(* PLC project Unnamed, Unknown Unnamed 1 *)
(* stored: creationDateTime 2024-02-27T18:06:15, modificationDateTime 2024-02-27T18:24:05 *)

PROGRAM Example

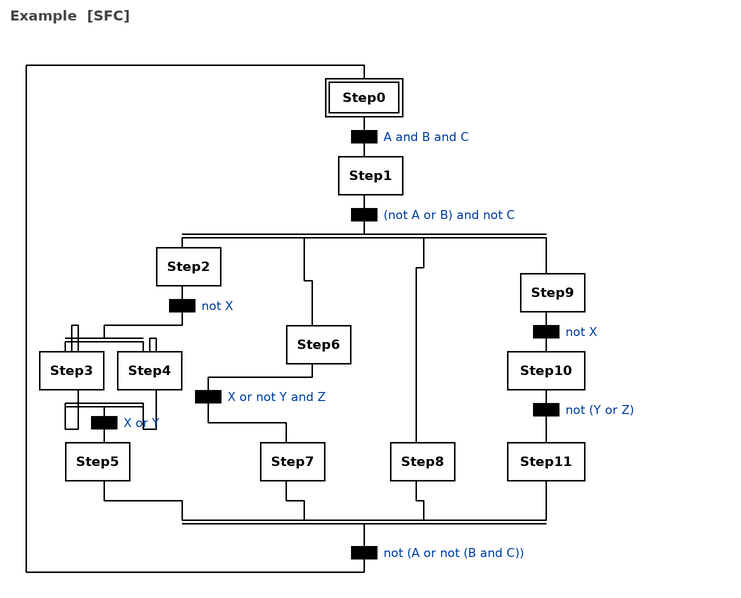
INITIAL_STEP Step0:
END_STEP
TRANSITION FROM Step0 TO Step1
  := A and B and C;
END_TRANSITION
STEP Step1:
END_STEP
TRANSITION FROM Step1 TO (Step2, Step6, Step8, Step9)
  := (not A or B) and not C;
END_TRANSITION
STEP Step2:
END_STEP
TRANSITION FROM Step2 TO (Step3, Step4)
  := not X;
END_TRANSITION
STEP Step9:
END_STEP
TRANSITION FROM Step9 TO Step10
  := not X;
END_TRANSITION
STEP Step6:
END_STEP
TRANSITION FROM Step6 TO Step7
  := X or not Y and Z;
END_TRANSITION
STEP Step3:
END_STEP
TRANSITION FROM (Step3, Step4) TO Step5
  := X or Y;
END_TRANSITION
STEP Step4:
END_STEP
STEP Step10:
END_STEP
TRANSITION FROM Step10 TO Step11
  := not (Y or Z);
END_TRANSITION
STEP Step5:
END_STEP
TRANSITION FROM (Step5, Step7, Step8, Step11) TO Step0
  := not (A or not (B and C));
END_TRANSITION
STEP Step7:
END_STEP
STEP Step8:
END_STEP
STEP Step11:
END_STEP
END_PROGRAM

CONFIGURATION Config0
  RESOURCE Res0 ON PLC
    TASK task0(INTERVAL := T#20ms, PRIORITY := 0);
    PROGRAM instance0 WITH task0 : Example;
  END_RESOURCE
END_CONFIGURATION
